{attribute 'GeneratedUsingTerminal: EK1100-0000-0018'}
{attribute addProperty BoxType "EK1100-0000-0018"}
{attribute addProperty Id "Beckhoff_EJ9xxxEK1122Beckhoff_EJ9xxxEK1122_C80E1DB32A_0001_EJ9001_0000_0016EJ9001_1FC0878B2A_0002_EJ9505_0000_0016EJ9505_19A4723D6A_0003_EJ9576_0000_0018EJ9576_6D7359CA28A_0004_EJ9576_0000_0019EJ9576_85AB580429A_0005_EJ9576_0000_0020EJ9576_1017F4A528A_0006_EJ9576_0000_0022EJ9576_C42142C629A_0007_EJ9400_0000EJ9400_B5091FDC0A_0008_EJ9404_0000EJ9404_A60D69000"}
{attribute addProperty CRC "1116610066"}
{attribute addProperty Size "124"}
TYPE Beckhoff_EJ9xxx_428E1E12 EXTENDS EK1100_1FC0878B :
STRUCT
	{attribute addProperty Name "Beckhoff EJ9xxxEK1122"}
	{attribute addProperty PreviousPort "Beckhoff EJ9xxx : B"}
	Beckhoff_EJ9xxxEK1122 : Beckhoff_EJ9xxxEK1122_C80E1DB3;
	{attribute addProperty Name "A_0001(EJ9001-0000-0016)"}
	{attribute addProperty PreviousPort "Beckhoff EJ9xxxEK1122 : C"}
	A_0001_EJ9001_0000_0016 : EJ9001_1FC0878B;
	{attribute addProperty Name "A_0002(EJ9505-0000-0016)"}
	{attribute addProperty PreviousPort "A_0001(EJ9001-0000-0016) : B"}
	A_0002_EJ9505_0000_0016 : EJ9505_19A4723D;
	{attribute addProperty Name "A_0003(EJ9576-0000-0018)"}
	{attribute addProperty PreviousPort "A_0002(EJ9505-0000-0016) : B"}
	A_0003_EJ9576_0000_0018 : EJ9576_6D7359CA;
	{attribute addProperty Name "A_0004(EJ9576-0000-0019)"}
	{attribute addProperty PreviousPort "A_0003(EJ9576-0000-0018) : B"}
	A_0004_EJ9576_0000_0019 : EJ9576_85AB5804;
	{attribute addProperty Name "A_0005(EJ9576-0000-0020)"}
	{attribute addProperty PreviousPort "A_0004(EJ9576-0000-0019) : B"}
	A_0005_EJ9576_0000_0020 : EJ9576_1017F4A5;
	{attribute addProperty Name "A_0006(EJ9576-0000-0022)"}
	{attribute addProperty PreviousPort "A_0005(EJ9576-0000-0020) : B"}
	A_0006_EJ9576_0000_0022 : EJ9576_C42142C6;
	{attribute addProperty Name "A_0007 (EJ9400-0000)"}
	{attribute addProperty PreviousPort "A_0006(EJ9576-0000-0022) : B"}
	A_0007_EJ9400_0000 : EJ9400_B5091FDC;
	{attribute addProperty Name "A_0008 (EJ9404-0000)"}
	{attribute addProperty PreviousPort "A_0006(EJ9576-0000-0022) : B"}
	A_0008_EJ9404_0000 : EJ9404_A60D6900;
END_STRUCT
END_TYPE

(* stored: Version 1.2.0.0, ProductVersion 3.1.4024.9
   DUT Beckhoff_EJ9xxx_428E1E12: Id {cfa99c03-6786-40f5-8f25-1043fbbbaa5c} *)
